FUNCTION_BLOCK PUBLIC FB_Pizza
VAR
	_PizzaState: INT;
	tonPizzaTimer : TON;
END_VAR

METHOD addCheese
VAR_INPUT
END_VAR
// Abstract Method
END_METHOD

METHOD addMeat
VAR_INPUT
END_VAR
//Abstract Method
END_METHOD

METHOD addVegetables : BOOL
VAR_INPUT
END_VAR
//Abstract Method
END_METHOD

METHOD bakePizza
VAR_INPUT
END_VAR
ADSLOGSTR( msgCtrlMask := ADSLOG_MSGTYPE_WARN,
        	msgFmtStr := 'Pizza is in the oven, please wait...', '');
END_METHOD

METHOD boxPizza
VAR_INPUT
END_VAR
ADSLOGSTR( msgCtrlMask := ADSLOG_MSGTYPE_WARN,
        	msgFmtStr := 'Pizza Boxed and Ready!!!', '');
END_METHOD

METHOD customerWantsCheese : BOOL
VAR_INPUT
END_VAR
customerWantsCheese := FALSE;
END_METHOD

METHOD customerWantsMeat : BOOL
VAR_INPUT
END_VAR
customerWantsMeat := FALSE;
END_METHOD

METHOD customerWantsVegetables : BOOL
VAR_INPUT
END_VAR
customerWantsVegetables := FALSE;
END_METHOD

METHOD FINAL makePizza
VAR_IN_OUT
	bExecute: BOOL;
END_VAR
CASE _PizzaState OF
	0: // Mandatory
		tonPizzaTimer(IN := bExecute, PT := T#2S); 
		IF tonPizzaTimer.Q THEN
			tonPizzaTimer(IN := FALSE, PT := T#2S); 
			bExecute := FALSE;
			rollDough();
			_PizzaState := 10;
		END_IF
		
	10: // Optional
		tonPizzaTimer(IN := TRUE, PT := T#2S); 
		IF tonPizzaTimer.Q THEN
			tonPizzaTimer(IN := FALSE, PT := T#2S); 
			IF(customerWantsCheese()) THEN
				addCheese();
			END_IF
			_PizzaState := 20;
		END_IF
		
	20: // Optional
		tonPizzaTimer(IN := TRUE, PT := T#2S); 
		IF tonPizzaTimer.Q THEN
			tonPizzaTimer(IN := FALSE, PT := T#2S); 
			IF(customerWantsMeat()) THEN
				addMeat();
			END_IF
			_PizzaState := 30;
		END_IF
		
	30: // Optional
		tonPizzaTimer(IN := TRUE, PT := T#2S); 
		IF tonPizzaTimer.Q THEN
			tonPizzaTimer(IN := FALSE, PT := T#2S); 
			IF(customerWantsVegetables()) THEN
				addVegetables();
			END_IF
			_PizzaState := 40;
		END_IF
		
	40: // Mandatory
		tonPizzaTimer(IN := TRUE, PT := T#2S);
 
		IF tonPizzaTimer.Q THEN
			tonPizzaTimer(IN := FALSE, PT := T#2S); 
			bakePizza();
			_PizzaState := 100;
		END_IF
		
	100:// Mandatory
		tonPizzaTimer(IN := TRUE, PT := T#2S); 
		
		IF tonPizzaTimer.Q THEN
			tonPizzaTimer(IN := FALSE, PT := T#2S); 
			boxPizza();
			_PizzaState := 0;
		END_IF
END_CASE
END_METHOD

METHOD rollDough
VAR_INPUT
END_VAR
ADSLOGSTR( msgCtrlMask := ADSLOG_MSGTYPE_WARN,
        	msgFmtStr := 'Rolling the Pizza Dough...', '');
END_METHOD

END_FUNCTION_BLOCK

(* stored: Version 1.1.0.1, ProductVersion 3.1.4024.12
   POU FB_Pizza: Id {4288fbe1-b507-4b53-980c-9e831d454702}, SpecialFunc None
   Method addCheese: Id {40c44adc-b934-41ec-97b9-4368975bc2f1}
   Method addMeat: Id {119b64f5-1788-467d-a213-c91d3435f9b9}
   Method addVegetables: Id {a0c4cca2-3178-4753-8594-fe871f75695c}
   Method bakePizza: Id {7b656edb-be36-4ff3-865d-b675da4cf248}
   Method boxPizza: Id {2f6381b0-8330-4e03-823e-93846c3ec2d1}
   Method customerWantsCheese: Id {7b637df3-3e0d-4785-a9d7-77c8387ccfc9}
   Method customerWantsMeat: Id {a5e9f7aa-0b61-4c6d-830f-4fe33cbd665e}
   Method customerWantsVegetables: Id {55a131b3-afac-4a8b-b480-9dc21f72edfa}
   Method makePizza: Id {c8d5e093-559d-4613-80fd-868bbbf84c5d}
   Method rollDough: Id {6151d24d-07a7-4f0e-a1a4-00165f91a29a} *)
